// SIMATIC S7-200 project (STEP 7-Micro/WIN), CPU 224XP REL 02.01

SYMBOL_TABLE USUARIO1
MARCHA           I0.0
LAMPARA_1        Q0.0
LAMPARA_2        Q0.1
END_SYMBOL_TABLE

ORGANIZATION_BLOCK PRINCIPAL:OB1
TITLE=COMENTARIOS DEL PROGRAMA
BEGIN
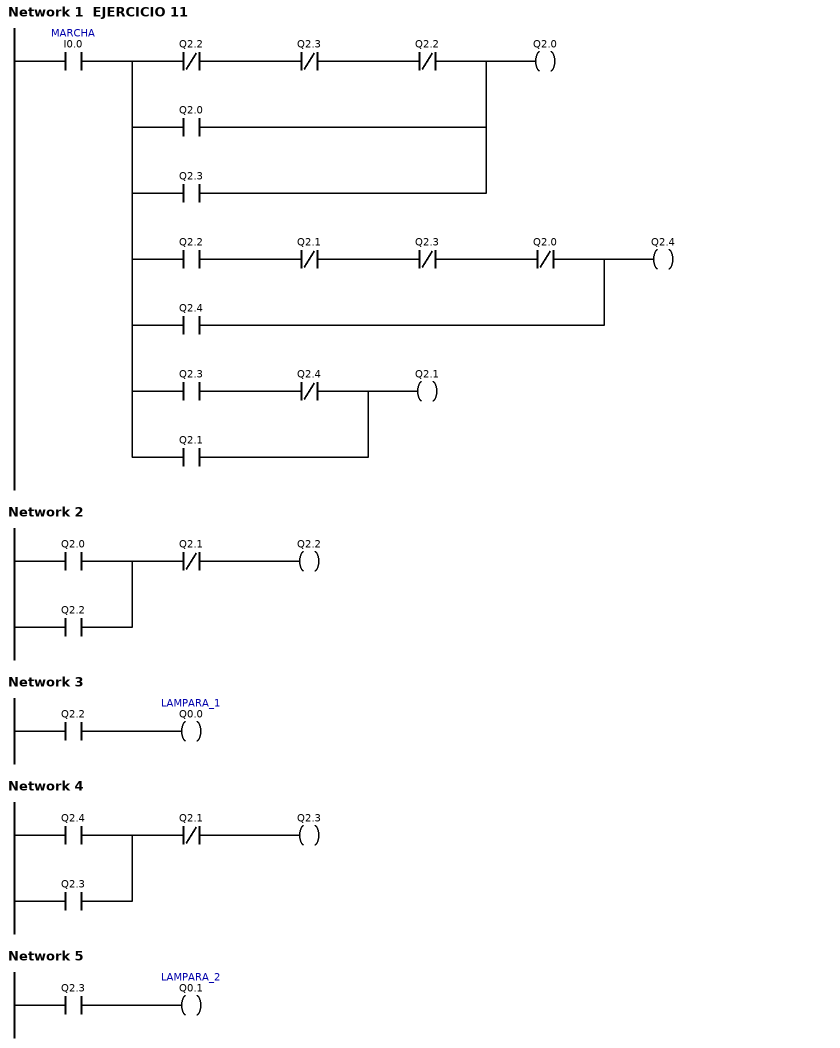
Network 1 // EJERCICIO 11 
LD     MARCHA:I0.0
LPS
LDN    Q2.2
AN     Q2.3
AN     Q2.2
O      Q2.0
O      Q2.3
ALD
=      Q2.0
LRD
LD     Q2.2
AN     Q2.1
AN     Q2.3
AN     Q2.0
O      Q2.4
ALD
=      Q2.4
LPP
LD     Q2.3
AN     Q2.4
O      Q2.1
ALD
=      Q2.1
Network 2
LD     Q2.0
O      Q2.2
AN     Q2.1
=      Q2.2
Network 3
LD     Q2.2
=      LAMPARA_1:Q0.0
Network 4
LD     Q2.4
O      Q2.3
AN     Q2.1
=      Q2.3
Network 5
LD     Q2.3
=      LAMPARA_2:Q0.1
END_ORGANIZATION_BLOCK
